Universal Robots PolyScope program: 1exBlink.urp

Program 1exBlink (installation=default directory=/home/ur/ursim-current/programs createdIn=5.11.8.1010444 lastSavedIn=5.11.8.1010444 robotSerialNumber=20195399999)
Calibrated DH parameters: a=[0, -0.24355, -0.2132, 0, 0, 0]; d=[0.15185, 0, 0, 0.13105, 0.08535, 0.0921]; alpha=[1.570796, 0, 0, 1.570796, -1.570796, 0]; deltaTheta=[0, 0, 0, 0, 0, 0]
BeforeStart
  Script file /home/ur/ursim-current/programs/Script/1_Ex_Led_blik.script
    | def BlinkLed(LED):
    | 	sleep(0.1)
    | 	set_digital_out(LED,True)
    | 	sleep(1.0)
    | 	set_digital_out(LED,False)
    | 	sleep(1.0)
    | end
Robot Program (runOnlyOnce=false)
  Script: BlinkLed(1)
